PROGRAM Stn055_41_StorageBypassMainMergePrestopRed
VAR
	{attribute 'TcLinkToOSO' := '.iPuckPresent    :=  <0,1,3>TIIB[N72S00 (AL1332)]^N72S05 (AL2341)^TxPDO^input byte 0;
								 .iBufferFull   :=  <0,1,3>TIIB[N72S00 (AL1332)]^N72S05 (AL2341)^TxPDO^input byte 2;
								 .oStopLower   :=  <0,1,4>TIIB[N72S00 (AL1332)]^N72S02 (EX260)^RxPDO^output byte 2'}
	fbConvStop: FB_ConvStop;
	
END_VAR

//  This code instantiates a component that is implimented as a common function block
//    Note that I/O is linked directly to I/O variables inside the named instance

gStn055_41_StorageBypassMainMergePrestopRed.ConvRunning := gConsumed_SafetyInterfaceConv.MtrRunning.Enc062Mtr04;

fbConvStop(
	pStn := ADR(gStn055),
	pCmp := ADR(gStn055_41_StorageBypassMainMergePrestopRed),
	pUpstreamStop := 0,
	pStateTraceBuffer := ADR(gStn055_StateTraceBuffer),
	pStateTraceFifo := ADR(gStn055_StateTraceFifo),
	pStats := ADR(gStn055_02_Stats));

END_PROGRAM

(* stored: Version 1.1.0.1, ProductVersion 3.1.4024.6
   POU Stn055_41_StorageBypassMainMergePrestopRed: Id {f19ee35f-02ee-48d5-bc75-ccb3e68cd9be}, SpecialFunc None *)
